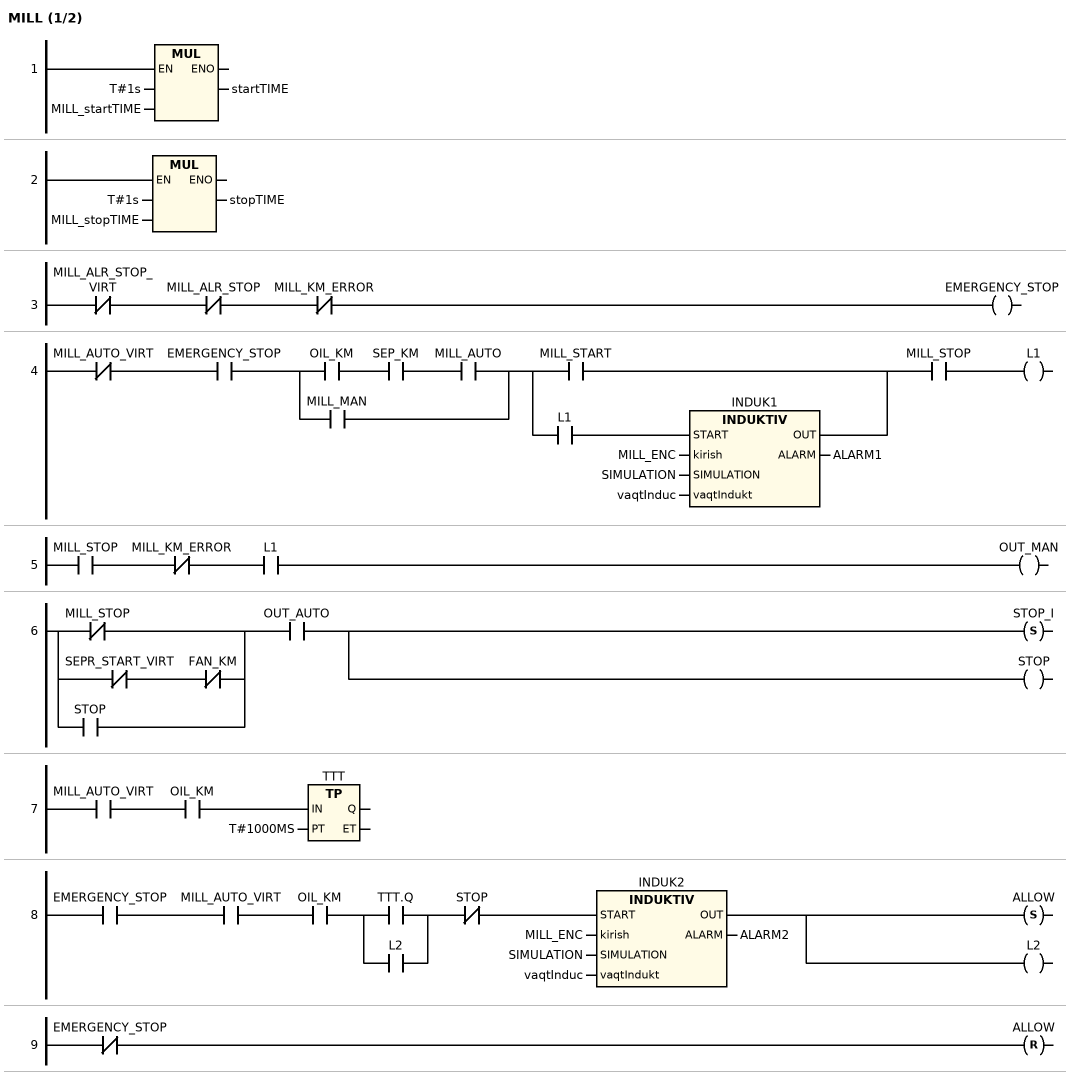
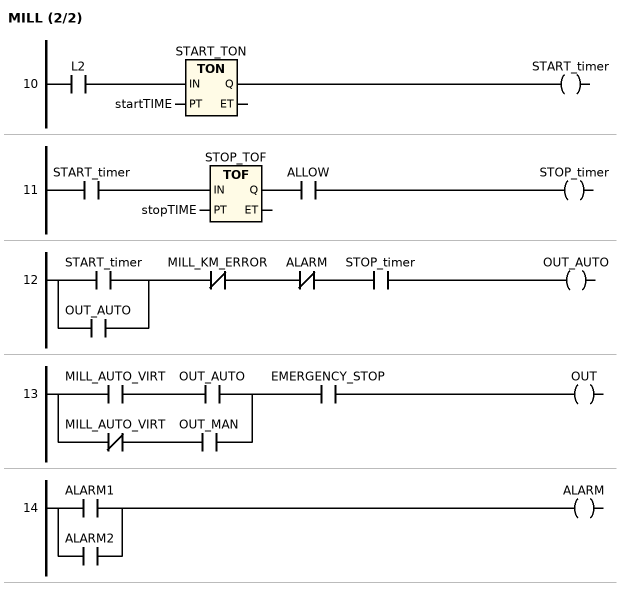
_LD_ (* Ladder Diagram *)
NETWORK 1
	*
		EN --- MUL(T#1s, MILL_startTIME) => startTIME
NETWORK 2
	*
		EN --- MUL(T#1s, MILL_stopTIME) => stopTIME
NETWORK 3
	[/MILL_ALR_STOP_VIRT] - [/MILL_ALR_STOP] - [/MILL_KM_ERROR] --- (EMERGENCY_STOP)
NETWORK 4
	[/MILL_AUTO_VIRT] - [EMERGENCY_STOP] - { [OIL_KM] - [SEP_KM] - [MILL_AUTO] | [MILL_MAN] } - { [MILL_START] | [L1] - INDUK1:INDUKTIV(START: *, kirish: MILL_ENC, SIMULATION: SIMULATION, vaqtIndukt: vaqtInduc, ALARM => ALARM1) } - [MILL_STOP] --- (L1)
NETWORK 5
	[MILL_STOP] - [/MILL_KM_ERROR] - [L1] --- (OUT_MAN)
NETWORK 6
	{ [/MILL_STOP] | [/SEPR_START_VIRT] - [/FAN_KM] | [STOP] } - [OUT_AUTO] --- (S STOP_I) (STOP)
NETWORK 7
	[MILL_AUTO_VIRT] - [OIL_KM] - TTT:TP(IN: *, PT: T#1000MS)
NETWORK 8
	[EMERGENCY_STOP] - [MILL_AUTO_VIRT] - [OIL_KM] - { [TTT.Q] | [L2] } - [/STOP] - INDUK2:INDUKTIV(START: *, kirish: MILL_ENC, SIMULATION: SIMULATION, vaqtIndukt: vaqtInduc, ALARM => ALARM2) --- (S ALLOW) (L2)
NETWORK 9
	[/EMERGENCY_STOP] --- (R ALLOW)
NETWORK 10
	[L2] - START_TON:TON(IN: *, PT: startTIME) --- (START_timer)
NETWORK 11
	[START_timer] - STOP_TOF:TOF(IN: *, PT: stopTIME) - [ALLOW] --- (STOP_timer)
NETWORK 12
	{ [START_timer] | [OUT_AUTO] } - [/MILL_KM_ERROR] - [/ALARM] - [STOP_timer] --- (OUT_AUTO)
NETWORK 13
	{ [MILL_AUTO_VIRT] - [OUT_AUTO] | [/MILL_AUTO_VIRT] - [OUT_MAN] } - [EMERGENCY_STOP] --- (OUT)
NETWORK 14
	{ [ALARM1] | [ALARM2] } --- (ALARM)
_END_LD_
(* the same logic as Structured Text *)
(* Network 1 *)
startTIME := T#1s * MILL_startTIME;
(* Network 2 *)
stopTIME := T#1s * MILL_stopTIME;
(* Network 3 *)
EMERGENCY_STOP := NOT MILL_ALR_STOP_VIRT AND NOT MILL_ALR_STOP AND NOT MILL_KM_ERROR;
(* Network 4 *)
_p1 := NOT MILL_AUTO_VIRT AND EMERGENCY_STOP AND (OIL_KM AND SEP_KM AND MILL_AUTO OR MILL_MAN);
INDUK1(START := _p1 AND L1, kirish := MILL_ENC, SIMULATION := SIMULATION, vaqtIndukt := vaqtInduc);
ALARM1 := INDUK1.ALARM;
L1 := (_p1 AND MILL_START OR INDUK1.OUT) AND MILL_STOP;
(* Network 5 *)
OUT_MAN := MILL_STOP AND NOT MILL_KM_ERROR AND L1;
(* Network 6 *)
_p2 := (NOT MILL_STOP OR NOT SEPR_START_VIRT AND NOT FAN_KM OR STOP) AND OUT_AUTO;
IF _p2 THEN STOP_I := TRUE; END_IF;
STOP := _p2;
(* Network 7 *)
TTT(IN := MILL_AUTO_VIRT AND OIL_KM, PT := T#1000MS);
(* Network 8 *)
INDUK2(START := EMERGENCY_STOP AND MILL_AUTO_VIRT AND OIL_KM AND (TTT.Q OR L2) AND NOT STOP, kirish := MILL_ENC, SIMULATION := SIMULATION, vaqtIndukt := vaqtInduc);
ALARM2 := INDUK2.ALARM;
IF INDUK2.OUT THEN ALLOW := TRUE; END_IF;
L2 := INDUK2.OUT;
(* Network 9 *)
IF NOT EMERGENCY_STOP THEN ALLOW := FALSE; END_IF;
(* Network 10 *)
START_TON(IN := L2, PT := startTIME);
START_timer := START_TON.Q;
(* Network 11 *)
STOP_TOF(IN := START_timer, PT := stopTIME);
STOP_timer := STOP_TOF.Q AND ALLOW;
(* Network 12 *)
OUT_AUTO := (START_timer OR OUT_AUTO) AND NOT MILL_KM_ERROR AND NOT ALARM AND STOP_timer;
(* Network 13 *)
OUT := (MILL_AUTO_VIRT AND OUT_AUTO OR NOT MILL_AUTO_VIRT AND OUT_MAN) AND EMERGENCY_STOP;
(* Network 14 *)
ALARM := ALARM1 OR ALARM2;
END_FUNCTION_BLOCK

(* POU FAN, LD *)
FUNCTION_BLOCK FAN
VAR_INPUT
	EN : BOOL;
	MILL_ALR_STOP: BOOL;
	MILL_ALR_STOP_VIRT : BOOL;
	MILL_AUTO : BOOL;
	MILL_AUTO_VIRT : BOOL;
	MILL_MAN : BOOL;
	FAN_START : BOOL;
	VIBRATOR_T : BOOL;

	FAN_STOP : BOOL;
	MILL_KM : BOOL;

	FAN_KM_ERROR : BOOL;
	SEPR_START_VIRT : BOOL;
	FAN_startTIME : WORD;
	FAN_stopTIME : WORD;
END_VAR

VAR_OUTPUT
	OUT : BOOL;
	ALARM : BOOL;
END_VAR
VAR
	INDUK1: INDUKTIV;
	INDUK2: INDUKTIV;
	OUT_MAN: BOOL;
	OUT_AUTO: BOOL;
	START_TON : TON;
	STOP_TOF : TOF;
	startTIME : TIME;
	stopTIME : TIME;
	L1: BOOL;
	L2: BOOL;
	ES: BOOL;
	EMERGENCY_STOP: BOOL;
	ALARM1 : BOOL;
	ALARM2 : BOOL;

	STOP: BOOL;
	ALLOW: BOOL;
	START_timer: BOOL;
	STOP_timer: BOOL;
	TTT : TP;
END_VAR
VAR (* helpers for the ST form of the networks *)
	_p1 : BOOL;
END_VAR
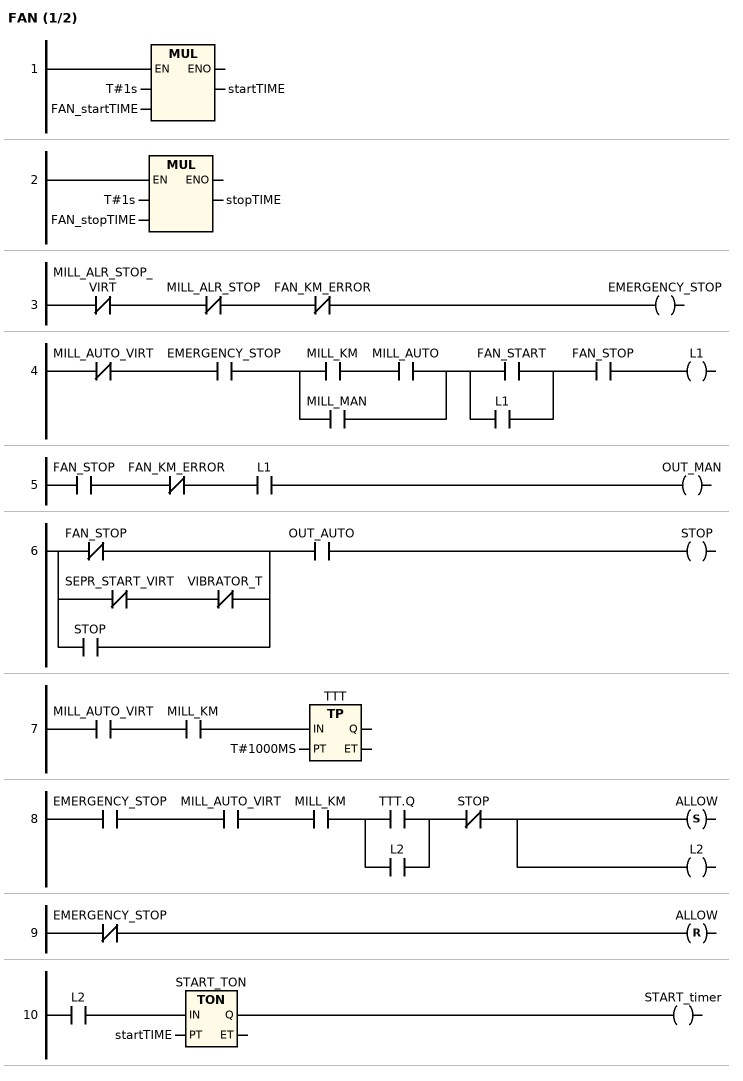
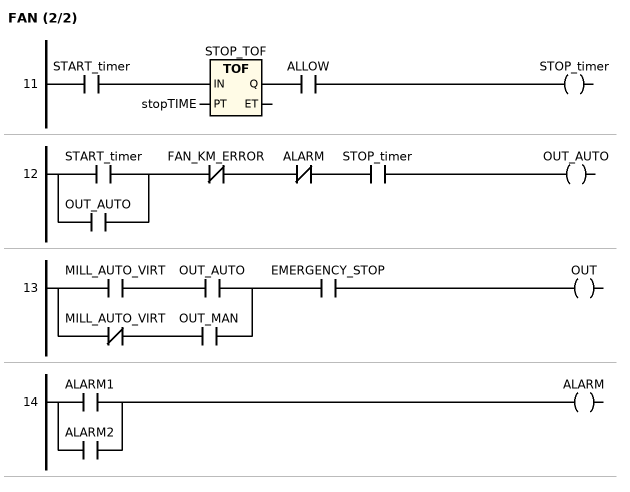
_LD_ (* Ladder Diagram *)
NETWORK 1
	*
		EN --- MUL(T#1s, FAN_startTIME) => startTIME
NETWORK 2
	*
		EN --- MUL(T#1s, FAN_stopTIME) => stopTIME
NETWORK 3
	[/MILL_ALR_STOP_VIRT] - [/MILL_ALR_STOP] - [/FAN_KM_ERROR] --- (EMERGENCY_STOP)
NETWORK 4
	[/MILL_AUTO_VIRT] - [EMERGENCY_STOP] - { [MILL_KM] - [MILL_AUTO] | [MILL_MAN] } - { [FAN_START] | [L1] } - [FAN_STOP] --- (L1)
NETWORK 5
	[FAN_STOP] - [/FAN_KM_ERROR] - [L1] --- (OUT_MAN)
NETWORK 6
	{ [/FAN_STOP] | [/SEPR_START_VIRT] - [/VIBRATOR_T] | [STOP] } - [OUT_AUTO] --- (STOP)
NETWORK 7
	[MILL_AUTO_VIRT] - [MILL_KM] - TTT:TP(IN: *, PT: T#1000MS)
NETWORK 8
	[EMERGENCY_STOP] - [MILL_AUTO_VIRT] - [MILL_KM] - { [TTT.Q] | [L2] } - [/STOP] --- (S ALLOW) (L2)
NETWORK 9
	[/EMERGENCY_STOP] --- (R ALLOW)
NETWORK 10
	[L2] - START_TON:TON(IN: *, PT: startTIME) --- (START_timer)
NETWORK 11
	[START_timer] - STOP_TOF:TOF(IN: *, PT: stopTIME) - [ALLOW] --- (STOP_timer)
NETWORK 12
	{ [START_timer] | [OUT_AUTO] } - [/FAN_KM_ERROR] - [/ALARM] - [STOP_timer] --- (OUT_AUTO)
NETWORK 13
	{ [MILL_AUTO_VIRT] - [OUT_AUTO] | [/MILL_AUTO_VIRT] - [OUT_MAN] } - [EMERGENCY_STOP] --- (OUT)
NETWORK 14
	{ [ALARM1] | [ALARM2] } --- (ALARM)
_END_LD_
(* the same logic as Structured Text *)
(* Network 1 *)
startTIME := T#1s * FAN_startTIME;
(* Network 2 *)
stopTIME := T#1s * FAN_stopTIME;
(* Network 3 *)
EMERGENCY_STOP := NOT MILL_ALR_STOP_VIRT AND NOT MILL_ALR_STOP AND NOT FAN_KM_ERROR;
(* Network 4 *)
L1 := NOT MILL_AUTO_VIRT AND EMERGENCY_STOP AND (MILL_KM AND MILL_AUTO OR MILL_MAN) AND (FAN_START OR L1) AND FAN_STOP;
(* Network 5 *)
OUT_MAN := FAN_STOP AND NOT FAN_KM_ERROR AND L1;
(* Network 6 *)
STOP := (NOT FAN_STOP OR NOT SEPR_START_VIRT AND NOT VIBRATOR_T OR STOP) AND OUT_AUTO;
(* Network 7 *)
TTT(IN := MILL_AUTO_VIRT AND MILL_KM, PT := T#1000MS);
(* Network 8 *)
_p1 := EMERGENCY_STOP AND MILL_AUTO_VIRT AND MILL_KM AND (TTT.Q OR L2) AND NOT STOP;
IF _p1 THEN ALLOW := TRUE; END_IF;
L2 := _p1;
(* Network 9 *)
IF NOT EMERGENCY_STOP THEN ALLOW := FALSE; END_IF;
(* Network 10 *)
START_TON(IN := L2, PT := startTIME);
START_timer := START_TON.Q;
(* Network 11 *)
STOP_TOF(IN := START_timer, PT := stopTIME);
STOP_timer := STOP_TOF.Q AND ALLOW;
(* Network 12 *)
OUT_AUTO := (START_timer OR OUT_AUTO) AND NOT FAN_KM_ERROR AND NOT ALARM AND STOP_timer;
(* Network 13 *)
OUT := (MILL_AUTO_VIRT AND OUT_AUTO OR NOT MILL_AUTO_VIRT AND OUT_MAN) AND EMERGENCY_STOP;
(* Network 14 *)
ALARM := ALARM1 OR ALARM2;
END_FUNCTION_BLOCK

(* POU CONV, LD *)
FUNCTION_BLOCK CONV
VAR_INPUT
	EN : BOOL;
	MILL_ALR_STOP: BOOL;
	MILL_ALR_STOP_VIRT : BOOL;
	MILL_AUTO : BOOL;
	MILL_AUTO_VIRT : BOOL;
	MILL_MAN : BOOL;
	CONV_START : BOOL;
	FAN_KM : BOOL;
	MILL_KM : BOOL;
	CONV_ENC : BOOL;
	CONV_STOP : BOOL;
	VIBRATOR_T : BOOL;
	CONV_KM_ERROR : BOOL;
	SIMULATION : BOOL := TRUE;
	MATER_FULL : BOOL;
	SEPR_START_VIRT : BOOL;
	vaqtInduc : WORD := 15;
END_VAR

VAR_OUTPUT
	OUT : BOOL;
	ALARM : BOOL;
END_VAR
VAR
	INDUK1: INDUKTIV;
	INDUK2: INDUKTIV;
	OUT_MAN: BOOL;
	OUT_AUTO: BOOL;
	START_TON : TON;
	STOP_TOF : TOF;
	startTIME : TIME;
	stopTIME : TIME;
	L1: BOOL;
	L2: BOOL;
	ES: BOOL;
	EMERGENCY_STOP: BOOL;
	ALARM1 : BOOL;
	ALARM2 : BOOL;

	STOP: BOOL;
	ALLOW: BOOL;
	START_timer: BOOL;
	STOP_timer: BOOL;
	TTT : TP;
END_VAR
VAR (* helpers for the ST form of the networks *)
	_p1 : BOOL;
END_VAR
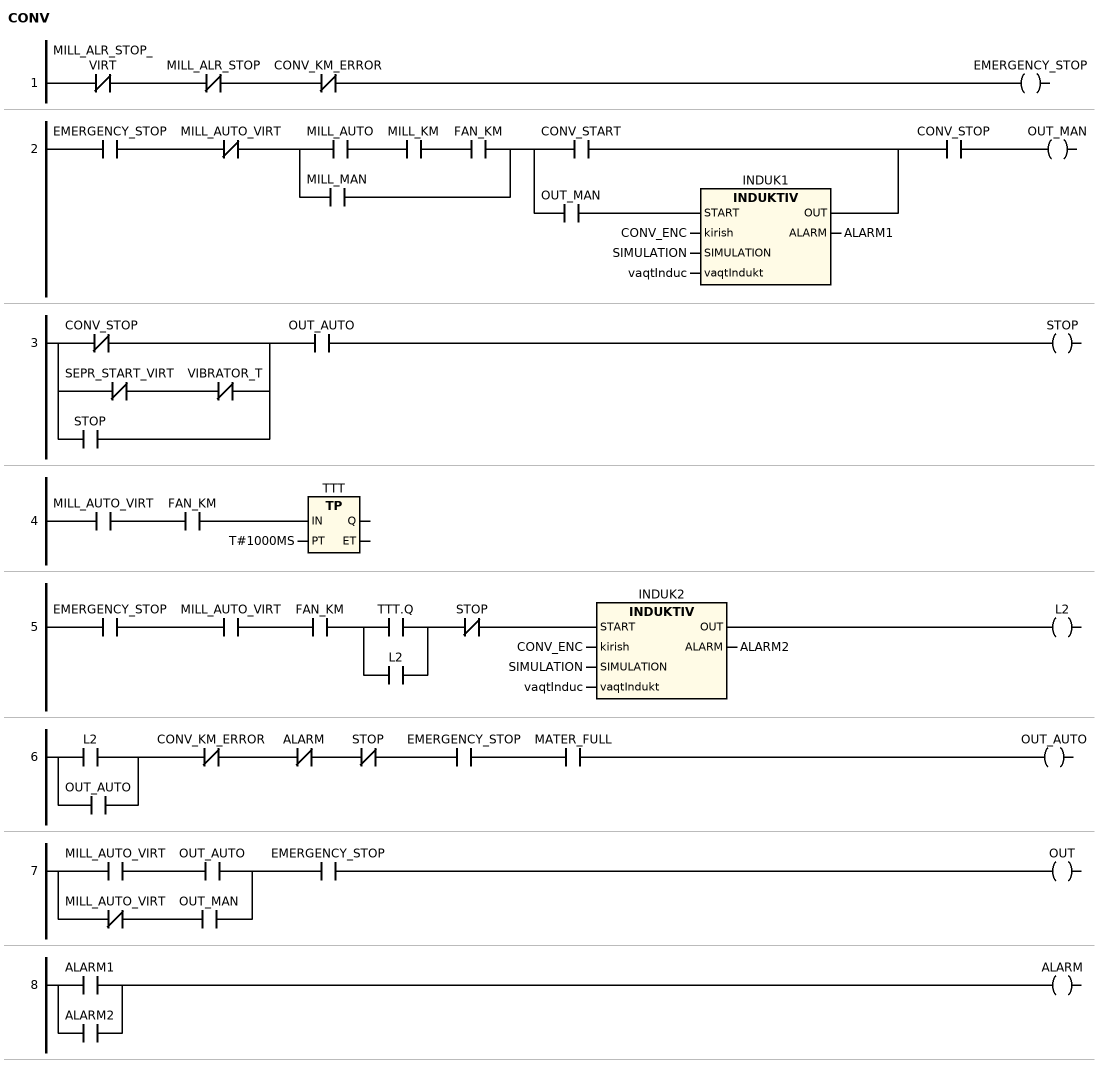
_LD_ (* Ladder Diagram *)
NETWORK 1
	[/MILL_ALR_STOP_VIRT] - [/MILL_ALR_STOP] - [/CONV_KM_ERROR] --- (EMERGENCY_STOP)
NETWORK 2
	[EMERGENCY_STOP] - [/MILL_AUTO_VIRT] - { [MILL_AUTO] - [MILL_KM] - [FAN_KM] | [MILL_MAN] } - { [CONV_START] | [OUT_MAN] - INDUK1:INDUKTIV(START: *, kirish: CONV_ENC, SIMULATION: SIMULATION, vaqtIndukt: vaqtInduc, ALARM => ALARM1) } - [CONV_STOP] --- (OUT_MAN)
NETWORK 3
	{ [/CONV_STOP] | [/SEPR_START_VIRT] - [/VIBRATOR_T] | [STOP] } - [OUT_AUTO] --- (STOP)
NETWORK 4
	[MILL_AUTO_VIRT] - [FAN_KM] - TTT:TP(IN: *, PT: T#1000MS)
NETWORK 5
	[EMERGENCY_STOP] - [MILL_AUTO_VIRT] - [FAN_KM] - { [TTT.Q] | [L2] } - [/STOP] - INDUK2:INDUKTIV(START: *, kirish: CONV_ENC, SIMULATION: SIMULATION, vaqtIndukt: vaqtInduc, ALARM => ALARM2) --- (L2)
NETWORK 6
	{ [L2] | [OUT_AUTO] } - [/CONV_KM_ERROR] - [/ALARM] - [/STOP] - [EMERGENCY_STOP] - [MATER_FULL] --- (OUT_AUTO)
NETWORK 7
	{ [MILL_AUTO_VIRT] - [OUT_AUTO] | [/MILL_AUTO_VIRT] - [OUT_MAN] } - [EMERGENCY_STOP] --- (OUT)
NETWORK 8
	{ [ALARM1] | [ALARM2] } --- (ALARM)
_END_LD_
(* the same logic as Structured Text *)
(* Network 1 *)
EMERGENCY_STOP := NOT MILL_ALR_STOP_VIRT AND NOT MILL_ALR_STOP AND NOT CONV_KM_ERROR;
(* Network 2 *)
_p1 := EMERGENCY_STOP AND NOT MILL_AUTO_VIRT AND (MILL_AUTO AND MILL_KM AND FAN_KM OR MILL_MAN);
INDUK1(START := _p1 AND OUT_MAN, kirish := CONV_ENC, SIMULATION := SIMULATION, vaqtIndukt := vaqtInduc);
ALARM1 := INDUK1.ALARM;
OUT_MAN := (_p1 AND CONV_START OR INDUK1.OUT) AND CONV_STOP;
(* Network 3 *)
STOP := (NOT CONV_STOP OR NOT SEPR_START_VIRT AND NOT VIBRATOR_T OR STOP) AND OUT_AUTO;
(* Network 4 *)
TTT(IN := MILL_AUTO_VIRT AND FAN_KM, PT := T#1000MS);
(* Network 5 *)
INDUK2(START := EMERGENCY_STOP AND MILL_AUTO_VIRT AND FAN_KM AND (TTT.Q OR L2) AND NOT STOP, kirish := CONV_ENC, SIMULATION := SIMULATION, vaqtIndukt := vaqtInduc);
ALARM2 := INDUK2.ALARM;
L2 := INDUK2.OUT;
(* Network 6 *)
OUT_AUTO := (L2 OR OUT_AUTO) AND NOT CONV_KM_ERROR AND NOT ALARM AND NOT STOP AND EMERGENCY_STOP AND MATER_FULL;
(* Network 7 *)
OUT := (MILL_AUTO_VIRT AND OUT_AUTO OR NOT MILL_AUTO_VIRT AND OUT_MAN) AND EMERGENCY_STOP;
(* Network 8 *)
ALARM := ALARM1 OR ALARM2;
END_FUNCTION_BLOCK

(* POU ALARMS, LD *)
PROGRAM ALARMS
VAR
	tofELV: TON;
	tofSHNK3: TON;
	tofSHNK4: TON;
	tofSHNK_SKL_3: TON;
	tofSHNK_SKL_4: TON;
	tofSTAR_31: TON;
	tofSTAR_32: TON;
	tofSTAR_41: TON;
	tofSTAR_42: TON;
	tofSEPR_3: TON;
	tofSEPR_4: TON;
	tofOIL_3: TON;
	tofOIL_4: TON;
	tofMILL_3: TON;
	tofMILL_4: TON;
	tofFAN_3: TON;
	tofFAN_4: TON;
	tofCONV_3: TON;
	tofCONV_4: TON;
	tofVIB_3: TON;
	tofVIB_4: TON;

	vaqt : TIME := T#30S;
END_VAR
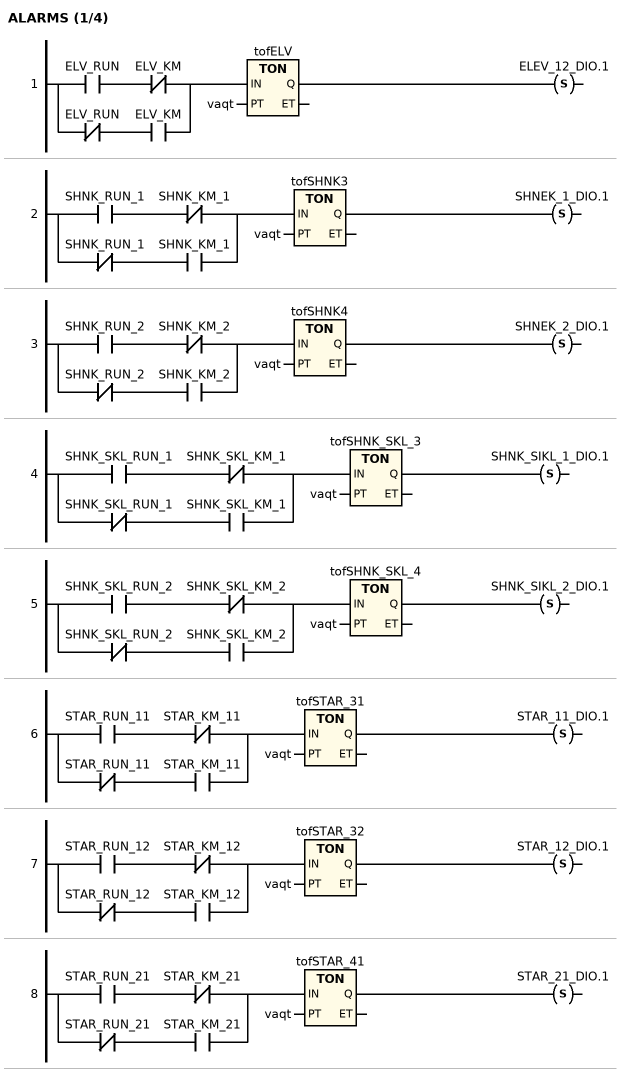
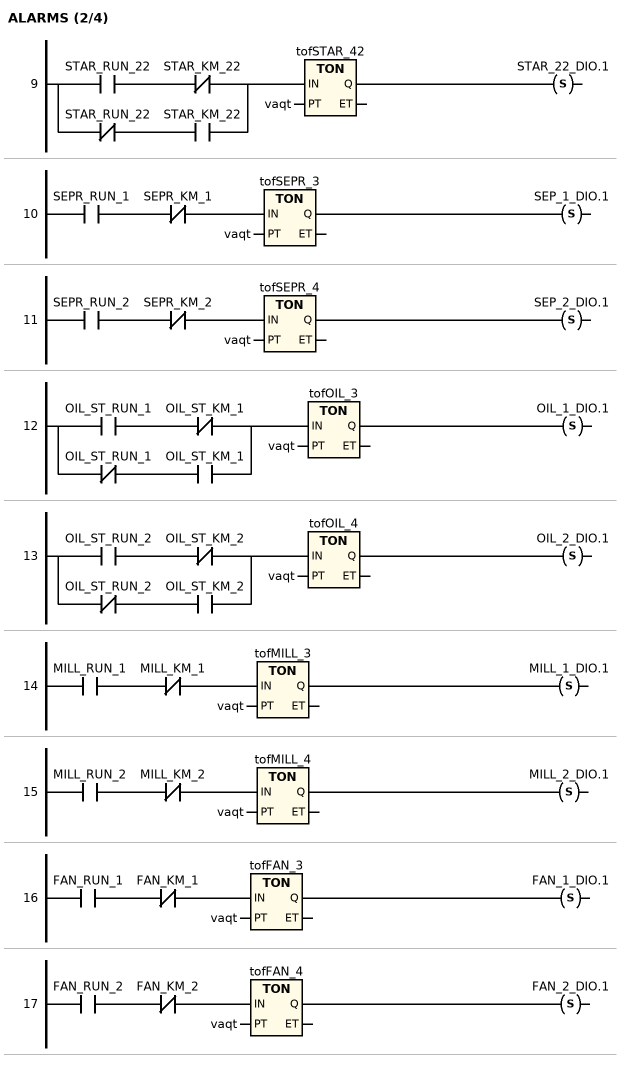
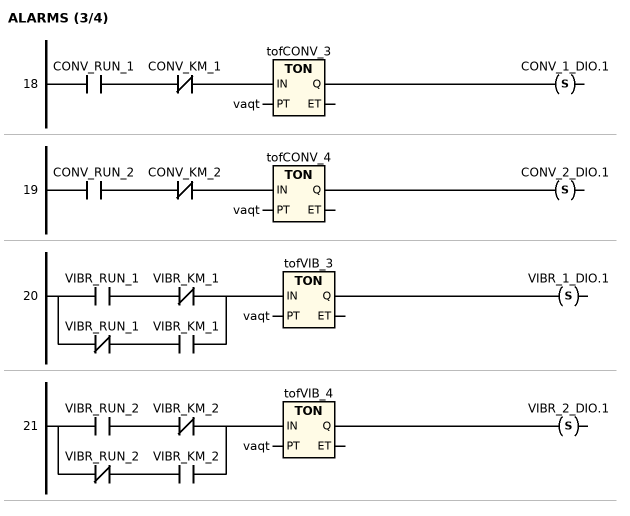
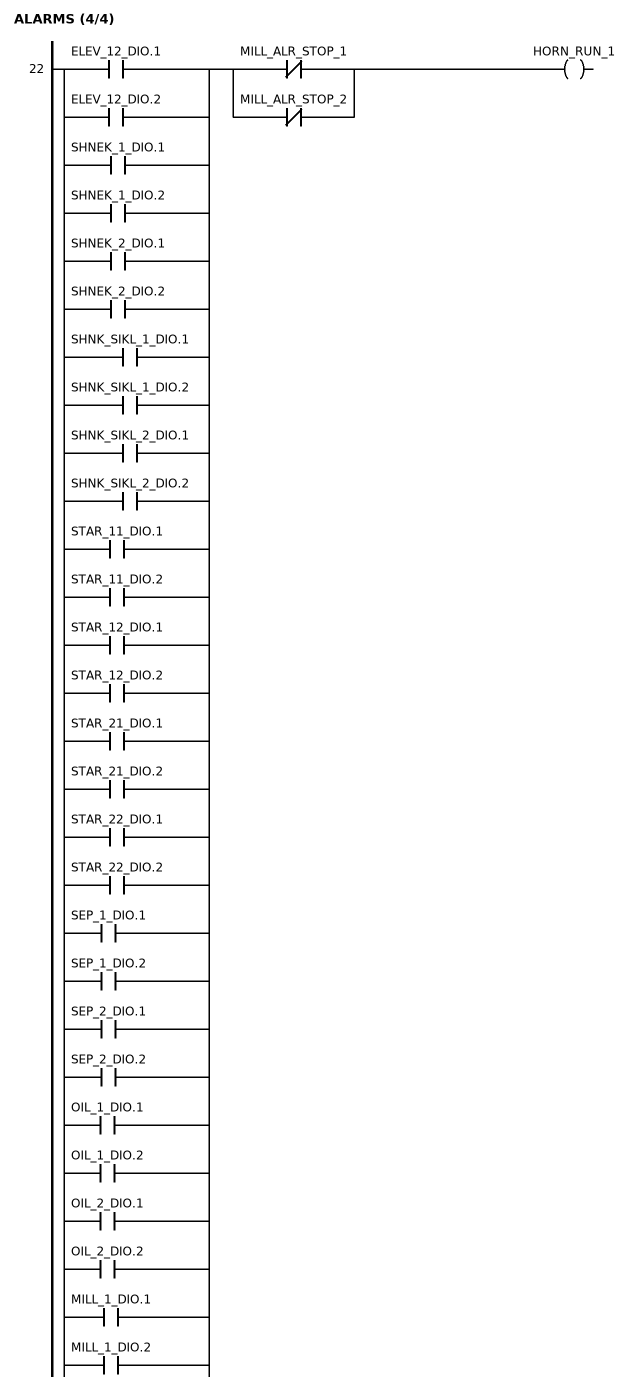
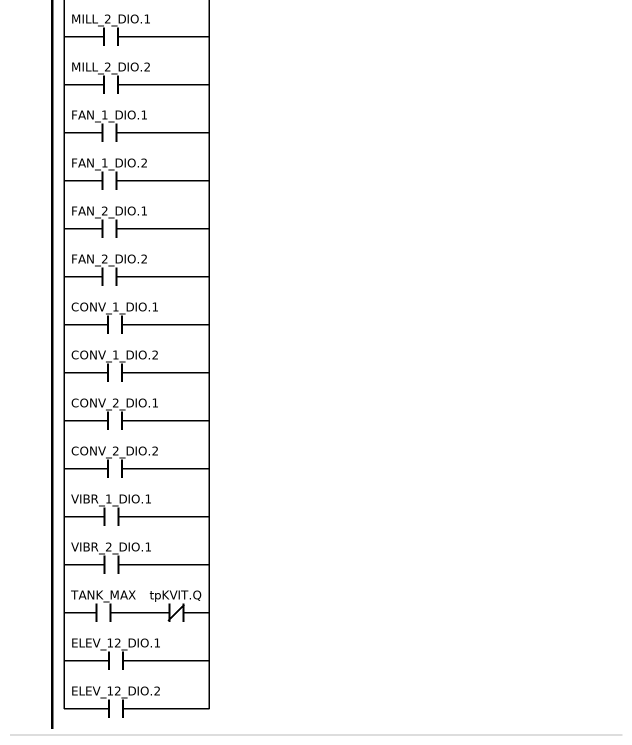
_LD_ (* Ladder Diagram *)
NETWORK 1
	{ [ELV_RUN] - [/ELV_KM] | [/ELV_RUN] - [ELV_KM] } - tofELV:TON(IN: *, PT: vaqt) --- (S ELEV_12_DIO.1)
NETWORK 2
	{ [SHNK_RUN_1] - [/SHNK_KM_1] | [/SHNK_RUN_1] - [SHNK_KM_1] } - tofSHNK3:TON(IN: *, PT: vaqt) --- (S SHNEK_1_DIO.1)
NETWORK 3
	{ [SHNK_RUN_2] - [/SHNK_KM_2] | [/SHNK_RUN_2] - [SHNK_KM_2] } - tofSHNK4:TON(IN: *, PT: vaqt) --- (S SHNEK_2_DIO.1)
NETWORK 4
	{ [SHNK_SKL_RUN_1] - [/SHNK_SKL_KM_1] | [/SHNK_SKL_RUN_1] - [SHNK_SKL_KM_1] } - tofSHNK_SKL_3:TON(IN: *, PT: vaqt) --- (S SHNK_SIKL_1_DIO.1)
NETWORK 5
	{ [SHNK_SKL_RUN_2] - [/SHNK_SKL_KM_2] | [/SHNK_SKL_RUN_2] - [SHNK_SKL_KM_2] } - tofSHNK_SKL_4:TON(IN: *, PT: vaqt) --- (S SHNK_SIKL_2_DIO.1)
NETWORK 6
	{ [STAR_RUN_11] - [/STAR_KM_11] | [/STAR_RUN_11] - [STAR_KM_11] } - tofSTAR_31:TON(IN: *, PT: vaqt) --- (S STAR_11_DIO.1)
NETWORK 7
	{ [STAR_RUN_12] - [/STAR_KM_12] | [/STAR_RUN_12] - [STAR_KM_12] } - tofSTAR_32:TON(IN: *, PT: vaqt) --- (S STAR_12_DIO.1)
NETWORK 8
	{ [STAR_RUN_21] - [/STAR_KM_21] | [/STAR_RUN_21] - [STAR_KM_21] } - tofSTAR_41:TON(IN: *, PT: vaqt) --- (S STAR_21_DIO.1)
NETWORK 9
	{ [STAR_RUN_22] - [/STAR_KM_22] | [/STAR_RUN_22] - [STAR_KM_22] } - tofSTAR_42:TON(IN: *, PT: vaqt) --- (S STAR_22_DIO.1)
NETWORK 10
	[SEPR_RUN_1] - [/SEPR_KM_1] - tofSEPR_3:TON(IN: *, PT: vaqt) --- (S SEP_1_DIO.1)
NETWORK 11
	[SEPR_RUN_2] - [/SEPR_KM_2] - tofSEPR_4:TON(IN: *, PT: vaqt) --- (S SEP_2_DIO.1)
NETWORK 12
	{ [OIL_ST_RUN_1] - [/OIL_ST_KM_1] | [/OIL_ST_RUN_1] - [OIL_ST_KM_1] } - tofOIL_3:TON(IN: *, PT: vaqt) --- (S OIL_1_DIO.1)
NETWORK 13
	{ [OIL_ST_RUN_2] - [/OIL_ST_KM_2] | [/OIL_ST_RUN_2] - [OIL_ST_KM_2] } - tofOIL_4:TON(IN: *, PT: vaqt) --- (S OIL_2_DIO.1)
NETWORK 14
	[MILL_RUN_1] - [/MILL_KM_1] - tofMILL_3:TON(IN: *, PT: vaqt) --- (S MILL_1_DIO.1)
NETWORK 15
	[MILL_RUN_2] - [/MILL_KM_2] - tofMILL_4:TON(IN: *, PT: vaqt) --- (S MILL_2_DIO.1)
NETWORK 16
	[FAN_RUN_1] - [/FAN_KM_1] - tofFAN_3:TON(IN: *, PT: vaqt) --- (S FAN_1_DIO.1)
NETWORK 17
	[FAN_RUN_2] - [/FAN_KM_2] - tofFAN_4:TON(IN: *, PT: vaqt) --- (S FAN_2_DIO.1)
NETWORK 18
	[CONV_RUN_1] - [/CONV_KM_1] - tofCONV_3:TON(IN: *, PT: vaqt) --- (S CONV_1_DIO.1)
NETWORK 19
	[CONV_RUN_2] - [/CONV_KM_2] - tofCONV_4:TON(IN: *, PT: vaqt) --- (S CONV_2_DIO.1)
NETWORK 20
	{ [VIBR_RUN_1] - [/VIBR_KM_1] | [/VIBR_RUN_1] - [VIBR_KM_1] } - tofVIB_3:TON(IN: *, PT: vaqt) --- (S VIBR_1_DIO.1)
NETWORK 21
	{ [VIBR_RUN_2] - [/VIBR_KM_2] | [/VIBR_RUN_2] - [VIBR_KM_2] } - tofVIB_4:TON(IN: *, PT: vaqt) --- (S VIBR_2_DIO.1)
NETWORK 22
	{ [ELEV_12_DIO.1] | [ELEV_12_DIO.2] | [SHNEK_1_DIO.1] | [SHNEK_1_DIO.2] | [SHNEK_2_DIO.1] | [SHNEK_2_DIO.2] | [SHNK_SIKL_1_DIO.1] | [SHNK_SIKL_1_DIO.2] | [SHNK_SIKL_2_DIO.1] | [SHNK_SIKL_2_DIO.2] | [STAR_11_DIO.1] | [STAR_11_DIO.2] | [STAR_12_DIO.1] | [STAR_12_DIO.2] | [STAR_21_DIO.1] | [STAR_21_DIO.2] | [STAR_22_DIO.1] | [STAR_22_DIO.2] | [SEP_1_DIO.1] | [SEP_1_DIO.2] | [SEP_2_DIO.1] | [SEP_2_DIO.2] | [OIL_1_DIO.1] | [OIL_1_DIO.2] | [OIL_2_DIO.1] | [OIL_2_DIO.2] | [MILL_1_DIO.1] | [MILL_1_DIO.2] | [MILL_2_DIO.1] | [MILL_2_DIO.2] | [FAN_1_DIO.1] | [FAN_1_DIO.2] | [FAN_2_DIO.1] | [FAN_2_DIO.2] | [CONV_1_DIO.1] | [CONV_1_DIO.2] | [CONV_2_DIO.1] | [CONV_2_DIO.2] | [VIBR_1_DIO.1] | [VIBR_2_DIO.1] | [TANK_MAX] - [/tpKVIT.Q] | [ELEV_12_DIO.1] | [ELEV_12_DIO.2] } - { [/MILL_ALR_STOP_1] | [/MILL_ALR_STOP_2] } --- (HORN_RUN_1)
_END_LD_
(* the same logic as Structured Text *)
(* Network 1 *)
tofELV(IN := ELV_RUN AND NOT ELV_KM OR NOT ELV_RUN AND ELV_KM, PT := vaqt);
IF tofELV.Q THEN ELEV_12_DIO.1 := TRUE; END_IF;
(* Network 2 *)
tofSHNK3(IN := SHNK_RUN_1 AND NOT SHNK_KM_1 OR NOT SHNK_RUN_1 AND SHNK_KM_1, PT := vaqt);
IF tofSHNK3.Q THEN SHNEK_1_DIO.1 := TRUE; END_IF;
(* Network 3 *)
tofSHNK4(IN := SHNK_RUN_2 AND NOT SHNK_KM_2 OR NOT SHNK_RUN_2 AND SHNK_KM_2, PT := vaqt);
IF tofSHNK4.Q THEN SHNEK_2_DIO.1 := TRUE; END_IF;
(* Network 4 *)
tofSHNK_SKL_3(IN := SHNK_SKL_RUN_1 AND NOT SHNK_SKL_KM_1 OR NOT SHNK_SKL_RUN_1 AND SHNK_SKL_KM_1, PT := vaqt);
IF tofSHNK_SKL_3.Q THEN SHNK_SIKL_1_DIO.1 := TRUE; END_IF;
(* Network 5 *)
tofSHNK_SKL_4(IN := SHNK_SKL_RUN_2 AND NOT SHNK_SKL_KM_2 OR NOT SHNK_SKL_RUN_2 AND SHNK_SKL_KM_2, PT := vaqt);
IF tofSHNK_SKL_4.Q THEN SHNK_SIKL_2_DIO.1 := TRUE; END_IF;
(* Network 6 *)
tofSTAR_31(IN := STAR_RUN_11 AND NOT STAR_KM_11 OR NOT STAR_RUN_11 AND STAR_KM_11, PT := vaqt);
IF tofSTAR_31.Q THEN STAR_11_DIO.1 := TRUE; END_IF;
(* Network 7 *)
tofSTAR_32(IN := STAR_RUN_12 AND NOT STAR_KM_12 OR NOT STAR_RUN_12 AND STAR_KM_12, PT := vaqt);
IF tofSTAR_32.Q THEN STAR_12_DIO.1 := TRUE; END_IF;
(* Network 8 *)
tofSTAR_41(IN := STAR_RUN_21 AND NOT STAR_KM_21 OR NOT STAR_RUN_21 AND STAR_KM_21, PT := vaqt);
IF tofSTAR_41.Q THEN STAR_21_DIO.1 := TRUE; END_IF;
(* Network 9 *)
tofSTAR_42(IN := STAR_RUN_22 AND NOT STAR_KM_22 OR NOT STAR_RUN_22 AND STAR_KM_22, PT := vaqt);
IF tofSTAR_42.Q THEN STAR_22_DIO.1 := TRUE; END_IF;
(* Network 10 *)
tofSEPR_3(IN := SEPR_RUN_1 AND NOT SEPR_KM_1, PT := vaqt);
IF tofSEPR_3.Q THEN SEP_1_DIO.1 := TRUE; END_IF;
(* Network 11 *)
tofSEPR_4(IN := SEPR_RUN_2 AND NOT SEPR_KM_2, PT := vaqt);
IF tofSEPR_4.Q THEN SEP_2_DIO.1 := TRUE; END_IF;
(* Network 12 *)
tofOIL_3(IN := OIL_ST_RUN_1 AND NOT OIL_ST_KM_1 OR NOT OIL_ST_RUN_1 AND OIL_ST_KM_1, PT := vaqt);
IF tofOIL_3.Q THEN OIL_1_DIO.1 := TRUE; END_IF;
(* Network 13 *)
tofOIL_4(IN := OIL_ST_RUN_2 AND NOT OIL_ST_KM_2 OR NOT OIL_ST_RUN_2 AND OIL_ST_KM_2, PT := vaqt);
IF tofOIL_4.Q THEN OIL_2_DIO.1 := TRUE; END_IF;
(* Network 14 *)
tofMILL_3(IN := MILL_RUN_1 AND NOT MILL_KM_1, PT := vaqt);
IF tofMILL_3.Q THEN MILL_1_DIO.1 := TRUE; END_IF;
(* Network 15 *)
tofMILL_4(IN := MILL_RUN_2 AND NOT MILL_KM_2, PT := vaqt);
IF tofMILL_4.Q THEN MILL_2_DIO.1 := TRUE; END_IF;
(* Network 16 *)
tofFAN_3(IN := FAN_RUN_1 AND NOT FAN_KM_1, PT := vaqt);
IF tofFAN_3.Q THEN FAN_1_DIO.1 := TRUE; END_IF;
(* Network 17 *)
tofFAN_4(IN := FAN_RUN_2 AND NOT FAN_KM_2, PT := vaqt);
IF tofFAN_4.Q THEN FAN_2_DIO.1 := TRUE; END_IF;
(* Network 18 *)
tofCONV_3(IN := CONV_RUN_1 AND NOT CONV_KM_1, PT := vaqt);
IF tofCONV_3.Q THEN CONV_1_DIO.1 := TRUE; END_IF;
(* Network 19 *)
tofCONV_4(IN := CONV_RUN_2 AND NOT CONV_KM_2, PT := vaqt);
IF tofCONV_4.Q THEN CONV_2_DIO.1 := TRUE; END_IF;
(* Network 20 *)
tofVIB_3(IN := VIBR_RUN_1 AND NOT VIBR_KM_1 OR NOT VIBR_RUN_1 AND VIBR_KM_1, PT := vaqt);
IF tofVIB_3.Q THEN VIBR_1_DIO.1 := TRUE; END_IF;
(* Network 21 *)
tofVIB_4(IN := VIBR_RUN_2 AND NOT VIBR_KM_2 OR NOT VIBR_RUN_2 AND VIBR_KM_2, PT := vaqt);
IF tofVIB_4.Q THEN VIBR_2_DIO.1 := TRUE; END_IF;
(* Network 22 *)
HORN_RUN_1 := (ELEV_12_DIO.1 OR ELEV_12_DIO.2 OR SHNEK_1_DIO.1 OR SHNEK_1_DIO.2 OR SHNEK_2_DIO.1 OR SHNEK_2_DIO.2 OR SHNK_SIKL_1_DIO.1 OR SHNK_SIKL_1_DIO.2 OR SHNK_SIKL_2_DIO.1 OR SHNK_SIKL_2_DIO.2 OR STAR_11_DIO.1 OR STAR_11_DIO.2 OR STAR_12_DIO.1 OR STAR_12_DIO.2 OR STAR_21_DIO.1 OR STAR_21_DIO.2 OR STAR_22_DIO.1 OR STAR_22_DIO.2 OR SEP_1_DIO.1 OR SEP_1_DIO.2 OR SEP_2_DIO.1 OR SEP_2_DIO.2 OR OIL_1_DIO.1 OR OIL_1_DIO.2 OR OIL_2_DIO.1 OR OIL_2_DIO.2 OR MILL_1_DIO.1 OR MILL_1_DIO.2 OR MILL_2_DIO.1 OR MILL_2_DIO.2 OR FAN_1_DIO.1 OR FAN_1_DIO.2 OR FAN_2_DIO.1 OR FAN_2_DIO.2 OR CONV_1_DIO.1 OR CONV_1_DIO.2 OR CONV_2_DIO.1 OR CONV_2_DIO.2 OR VIBR_1_DIO.1 OR VIBR_2_DIO.1 OR TANK_MAX AND NOT tpKVIT.Q OR ELEV_12_DIO.1 OR ELEV_12_DIO.2) AND (NOT MILL_ALR_STOP_1 OR NOT MILL_ALR_STOP_2);
END_PROGRAM

(* POU RESET_ALRM, LD *)
PROGRAM RESET_ALRM
VAR
END_VAR
VAR (* helpers for the ST form of the networks *)
	_p1 : BOOL;
END_VAR
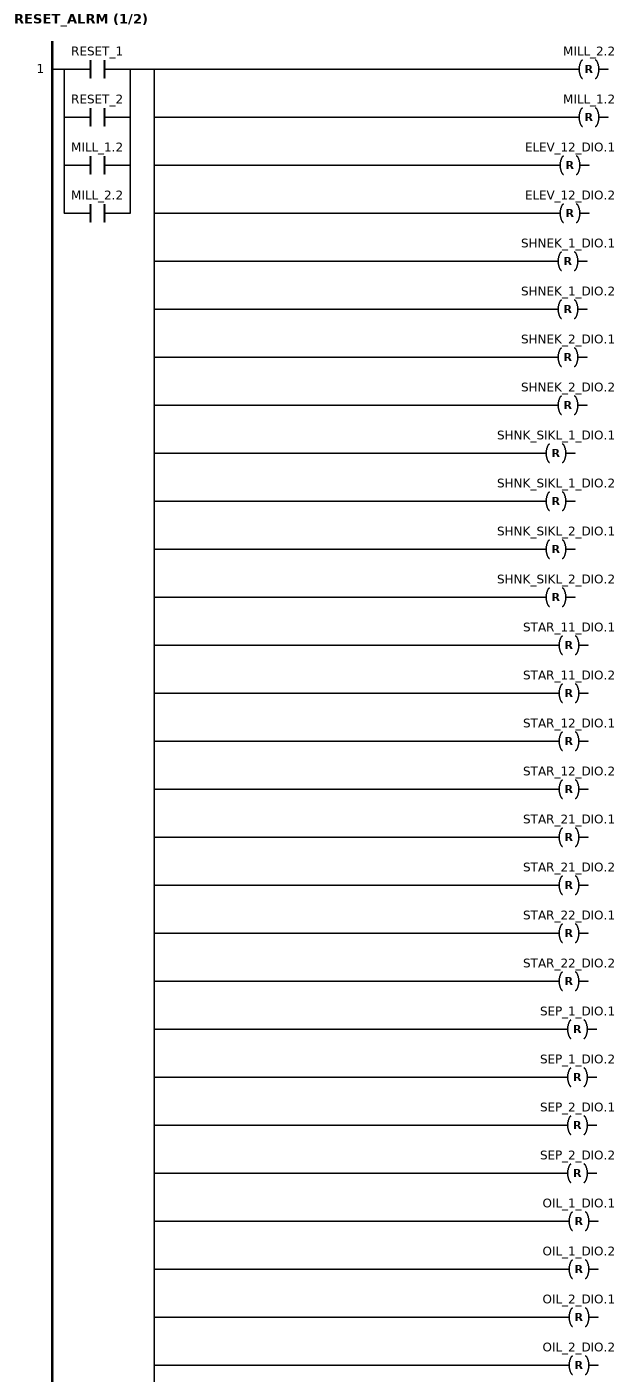
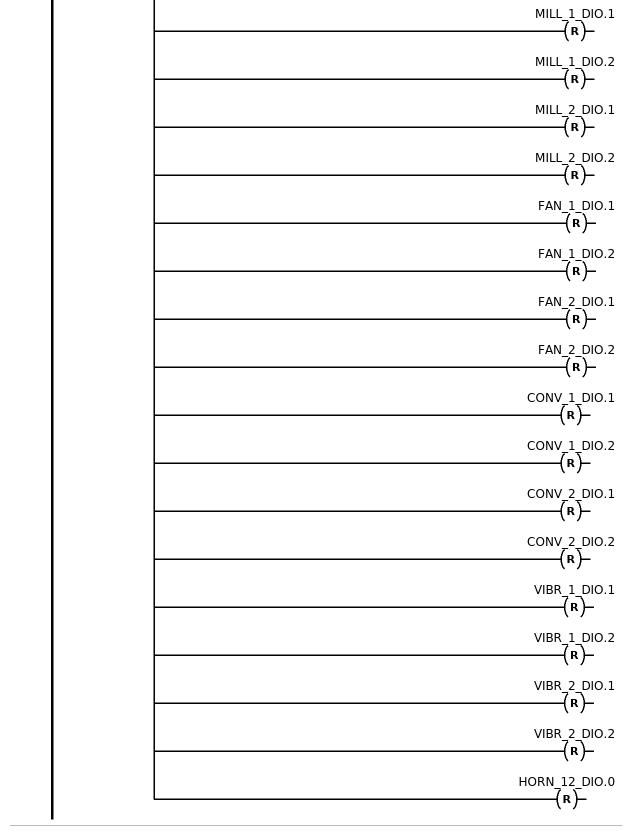
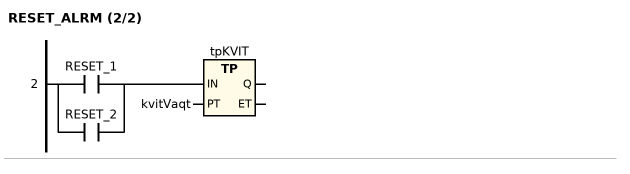
_LD_ (* Ladder Diagram *)
NETWORK 1
	{ [RESET_1] | [RESET_2] | [MILL_1.2] | [MILL_2.2] } --- (R MILL_2.2) (R MILL_1.2) (R ELEV_12_DIO.1) (R ELEV_12_DIO.2) (R SHNEK_1_DIO.1) (R SHNEK_1_DIO.2) (R SHNEK_2_DIO.1) (R SHNEK_2_DIO.2) (R SHNK_SIKL_1_DIO.1) (R SHNK_SIKL_1_DIO.2) (R SHNK_SIKL_2_DIO.1) (R SHNK_SIKL_2_DIO.2) (R STAR_11_DIO.1) (R STAR_11_DIO.2) (R STAR_12_DIO.1) (R STAR_12_DIO.2) (R STAR_21_DIO.1) (R STAR_21_DIO.2) (R STAR_22_DIO.1) (R STAR_22_DIO.2) (R SEP_1_DIO.1) (R SEP_1_DIO.2) (R SEP_2_DIO.1) (R SEP_2_DIO.2) (R OIL_1_DIO.1) (R OIL_1_DIO.2) (R OIL_2_DIO.1) (R OIL_2_DIO.2) (R MILL_1_DIO.1) (R MILL_1_DIO.2) (R MILL_2_DIO.1) (R MILL_2_DIO.2) (R FAN_1_DIO.1) (R FAN_1_DIO.2) (R FAN_2_DIO.1) (R FAN_2_DIO.2) (R CONV_1_DIO.1) (R CONV_1_DIO.2) (R CONV_2_DIO.1) (R CONV_2_DIO.2) (R VIBR_1_DIO.1) (R VIBR_1_DIO.2) (R VIBR_2_DIO.1) (R VIBR_2_DIO.2) (R HORN_12_DIO.0)
NETWORK 2
	{ [RESET_1] | [RESET_2] } - tpKVIT:TP(IN: *, PT: kvitVaqt)
_END_LD_
(* the same logic as Structured Text *)
(* Network 1 *)
_p1 := RESET_1 OR RESET_2 OR MILL_1.2 OR MILL_2.2;
IF _p1 THEN MILL_2.2 := FALSE; MILL_1.2 := FALSE; ELEV_12_DIO.1 := FALSE; ELEV_12_DIO.2 := FALSE; SHNEK_1_DIO.1 := FALSE; SHNEK_1_DIO.2 := FALSE; SHNEK_2_DIO.1 := FALSE; SHNEK_2_DIO.2 := FALSE; SHNK_SIKL_1_DIO.1 := FALSE; SHNK_SIKL_1_DIO.2 := FALSE; SHNK_SIKL_2_DIO.1 := FALSE; SHNK_SIKL_2_DIO.2 := FALSE; STAR_11_DIO.1 := FALSE; STAR_11_DIO.2 := FALSE; STAR_12_DIO.1 := FALSE; STAR_12_DIO.2 := FALSE; STAR_21_DIO.1 := FALSE; STAR_21_DIO.2 := FALSE; STAR_22_DIO.1 := FALSE; STAR_22_DIO.2 := FALSE; SEP_1_DIO.1 := FALSE; SEP_1_DIO.2 := FALSE; SEP_2_DIO.1 := FALSE; SEP_2_DIO.2 := FALSE; OIL_1_DIO.1 := FALSE; OIL_1_DIO.2 := FALSE; OIL_2_DIO.1 := FALSE; OIL_2_DIO.2 := FALSE; MILL_1_DIO.1 := FALSE; MILL_1_DIO.2 := FALSE; MILL_2_DIO.1 := FALSE; MILL_2_DIO.2 := FALSE; FAN_1_DIO.1 := FALSE; FAN_1_DIO.2 := FALSE; FAN_2_DIO.1 := FALSE; FAN_2_DIO.2 := FALSE; CONV_1_DIO.1 := FALSE; CONV_1_DIO.2 := FALSE; CONV_2_DIO.1 := FALSE; CONV_2_DIO.2 := FALSE; VIBR_1_DIO.1 := FALSE; VIBR_1_DIO.2 := FALSE; VIBR_2_DIO.1 := FALSE; VIBR_2_DIO.2 := FALSE; HORN_12_DIO.0 := FALSE; END_IF;
(* Network 2 *)
tpKVIT(IN := RESET_1 OR RESET_2, PT := kvitVaqt);
END_PROGRAM

(* POU TRANSLATE, ST *)
PROGRAM TRANSLATE
VAR
	CON1: A_CONVER;
	CON2: A_CONVER;
	CON3: MY_LIN_TRAFO;
	CON4: A_CONVER;
	CON5: MY_LIN_TRAFO;
	tonTank : TON;
	IN_MIN : REAL := 4;
	IN_MAX: REAL := 20;
	OUT_MIN_SEN : REAL := -10;
	OUT_MAX_SEN: REAL := 1;
	OUT_MIN_CUR : REAL := 0;
	OUT_MAX_CUR: REAL := 50;
END_VAR
freqTask();
MB_ANALOG();

hour_MOVE();


MV8();
MV16();
MV24();
MU32_OUT();
workHour();
TANK_12_DIO.0 := TANK_MIN;
TANK_12_DIO.1 := TANK_MIDL;
TANK_12_DIO.2 := TANK_MAX;
tonTank(IN := TANK_MAX_DI, PT := T#10s);
TANK_MAX := tonTank.Q;
END_PROGRAM
ACTION hour_MOVE:
CONV_1_stopTIME := CONV_1_stopTIME_W;
CONV_1_startTIME := CONV_1_startTIME_W;
FAN_1_stopTIME := FAN_1_stopTIME_W;
FAN_1_startTIME := FAN_1_startTIME_W;
MILL_1_stopTIME := MILL_1_stopTIME_W;
MILL_1_startTIME := MILL_1_startTIME_W;
SEP_1_stopTIME := SEP_1_stopTIME_W;
SEP_1_startTIME := SEP_1_startTIME_W;
CONV_2_stopTIME := CONV_2_stopTIME_W;
CONV_2_startTIME := CONV_2_startTIME_W;
FAN_2_stopTIME := FAN_2_stopTIME_W;
FAN_2_startTIME := FAN_2_startTIME_W;
MILL_2_stopTIME := MILL_2_stopTIME_W;
MILL_2_startTIME := MILL_2_startTIME_W;
SEP_2_stopTIME := SEP_2_stopTIME_W;
SEP_2_startTIME:= SEP_2_startTIME_W;
ELEV_12_stopTIME := ELEV_12_stopTIME_W;
ELEV_12_startTIME := ELEV_12_startTIME_W;
SHNEK_1_stopTIME := SHNEK_1_stopTIME_W;
SHNEK_2_stopTIME := SHNEK_2_stopTIME_W;
SHNEK_1_startTIME := SHNEK_1_startTIME_W;
SHNEK_2_startTIME := SHNEK_2_startTIME_W;
STAR_11_stopTIME := STAR_11_stopTIME_W;
STAR_11_startTIME := STAR_11_startTIME_W;
STAR_12_stopTIME := STAR_12_stopTIME_W;
STAR_12_startTIME := STAR_12_startTIME_W;
STAR_21_stopTIME := STAR_21_stopTIME_W;
STAR_21_startTIME := STAR_21_startTIME_W;
STAR_22_stopTIME := STAR_22_stopTIME_W;
STAR_22_startTIME := STAR_22_startTIME_W;
OIL_1_stopTIME := OIL_1_stopTIME_W;
OIL_1_startTIME := OIL_1_startTIME_W;
OIL_2_stopTIME := OIL_2_stopTIME_W;
OIL_2_startTIME := OIL_2_startTIME_W;
SHNK_SIKL_1_stopTIME := SHNK_SIKL_1_stopTIME_W;
SHNK_SIKL_1_startTIME := SHNK_SIKL_1_startTIME_W;
SHNK_SIKL_2_stopTIME := SHNK_SIKL_2_stopTIME_W;
SHNK_SIKL_2_startTIME := SHNK_SIKL_2_startTIME_W;
END_ACTION
ACTION MB_ANALOG:
ELEV_12_CURRENT := ELV_CURRENT_4;
SHNEK_2_CURRENT := SHNK_CURRENT_4;
FAN_2_SUCTION := MILL_SUCTION_4;
SHNEK_1_CURRENT := SHNK_CURRENT_3;
FAN_1_SUCTION := MILL_SUCTION_3;
END_ACTION
ACTION MU32_OUT:
MU01 := BOOL_TO_WORD(ELV_RUN) * 1000;
MU02 := BOOL_TO_WORD(SHNK_RUN_2) * 1000;
MU03 := BOOL_TO_WORD(SHNK_SKL_RUN_2) * 1000;
MU04 := BOOL_TO_WORD(STAR_RUN_21) * 1000;
MU05 := BOOL_TO_WORD(STAR_RUN_22) * 1000;
MU06 := BOOL_TO_WORD(SEPR_RUN_2) * 1000;
MU07 := BOOL_TO_WORD(OIL_ST_RUN_2) * 1000;
MU08 := BOOL_TO_WORD(MILL_RUN_2) * 1000;
MU09 := BOOL_TO_WORD(FAN_RUN_2) * 1000;
MU10 := BOOL_TO_WORD(CONV_RUN_2) * 1000;
MU11 := BOOL_TO_WORD(VIBR_RUN_2) * 1000;
MU12 := BOOL_TO_WORD(VALV_RUN_2) * 1000;
MU13 := BOOL_TO_WORD(HORN_RUN_2) * 1000;
(*
MU14 := BOOL_TO_WORD(m_out14) * 1000;
MU15 := BOOL_TO_WORD(m_out15) * 1000;
MU16 := BOOL_TO_WORD(m_out16) * 1000;
*)
MU17 := BOOL_TO_WORD(ELV_RUN) * 1000;
MU18 := BOOL_TO_WORD(SHNK_RUN_1) * 1000;
MU19 := BOOL_TO_WORD(SHNK_SKL_RUN_1) * 1000;
MU20 := BOOL_TO_WORD(STAR_RUN_11) * 1000;
MU21 := BOOL_TO_WORD(STAR_RUN_12) * 1000;
MU22 := BOOL_TO_WORD(SEPR_RUN_1) * 1000;
MU23 := BOOL_TO_WORD(OIL_ST_RUN_1) * 1000;
MU24 := BOOL_TO_WORD(MILL_RUN_1) * 1000;
MU25 := BOOL_TO_WORD(FAN_RUN_1) * 1000;
MU26 := BOOL_TO_WORD(CONV_RUN_1) * 1000;
MU27 := BOOL_TO_WORD(VIBR_RUN_1) * 1000;
MU28 := BOOL_TO_WORD(VALV_RUN_1) * 1000;
MU29 := BOOL_TO_WORD(HORN_RUN_1) * 1000;
(*
MU30 := BOOL_TO_WORD(m_out30) * 1000;
MU31 := BOOL_TO_WORD(m_out31) * 1000;
MU32 := BOOL_TO_WORD(m_out32) * 1000;
*)
END_ACTION
ACTION MV16:
ELEV_12_DIO.4			 := ELV_STOP_1	 		:= MV16_0.0;
SHNEK_1_DIO.4 			 := SHNK_STOP_1		 := MV16_0.1;
SHNK_SIKL_1_DIO.4		 :=  SHNK_SKL_STOP_1	 := MV16_0.2;
STAR_11_DIO.4			 := STAR_STOP_11		 := MV16_0.3;
STAR_12_DIO.4			 := STAR_STOP_12		 := MV16_0.4;
SEP_1_DIO.4 				 := SEPR_STOP_1		 := MV16_0.5;
OIL_1_DIO.4				 := OIL_ST_STOP_1		 := MV16_0.6;
MILL_1_DIO.4				 := MILL_STOP_1			 := MV16_0.7;
FAN_1_DIO.4				 := FAN_STOP_1			 := MV16_0.8;
CONV_1_DIO.4			 := CONV_STOP_1		 := MV16_0.9;
VIBR_1_DIO.4                     := VIBR_STOP_1			 := MV16_0.10;
(**********************)
ELEV_12_DIO.3			 := ELV_START_1			 := MV16_1.0;
SHNEK_1_DIO.3 			 := SHNK_START_1		 := MV16_1.1;
SHNK_SIKL_1_DIO.3		 := SHNK_SKL_START_1 := MV16_1.2;
STAR_11_DIO.3			 := STAR_START_11		 := MV16_1.3;
STAR_12_DIO.3			 := STAR_START_12		 := MV16_1.4;
SEP_1_DIO.3 				 := SEPR_START_1		 := MV16_1.5;
OIL_1_DIO.3				 := OIL_ST_START_1		 := MV16_1.6;
MILL_1_DIO.3				 := MILL_START_1		 := MV16_1.7;
FAN_1_DIO.3				 := FAN_START_1 			 := MV16_1.8;
CONV_1_DIO.3			 := CONV_START_1 		 := MV16_1.9;
VIBR_1_DIO.3                     := VIBR_START_1		 := MV16_1.10;
END_ACTION
ACTION MV24:
ELV_KM := MV24_0.0;
SHNK_KM_2 := MV24_0.1;
SHNK_SKL_KM_2 := MV24_0.2;
STAR_KM_21 := MV24_0.3;
STAR_KM_22 := MV24_0.4;
SEPR_KM_2 := MV24_0.5;
OIL_ST_KM_2 := MV24_0.6;
MILL_KM_2 := MV24_0.7;
MILL_2_DIO.8 := MATER_FULL_2 := MV24_0.8;
FAN_KM_2 := MV24_0.9;
CONV_KM_2 := MV24_0.10;
VIBR_KM_2 := MV24_0.11;
(*********
ELV_KM_3 := MV24_1.0;*)
SHNK_KM_1 := MV24_1.1;
SHNK_SKL_KM_1 := MV24_1.2;
STAR_KM_11 := MV24_1.3;
STAR_KM_12 := MV24_1.4;
SEPR_KM_1 := MV24_1.5;
OIL_ST_KM_1 := MV24_1.6;
MILL_KM_1 := MV24_1.7;
MILL_1_DIO.8 := MATER_FULL_1 := MV24_1.8;
FAN_KM_1 := MV24_1.9;
CONV_KM_1 := MV24_1.10;
VIBR_KM_1 := MV24_1.11;
END_ACTION
ACTION MV8:
ELV_STOP_2 := MV8_0.0;
SHNK_STOP_2 := MV8_0.1;
SHNK_SKL_STOP_2 := MV8_0.2;


STAR_21_DIO.4 			:= STAR_STOP_21 			:= MV8_0.3;
STAR_22_DIO.4 			:= STAR_STOP_22			 := MV8_0.4;
SEP_2_DIO.4 				 :=SEPR_STOP_2				 := MV8_0.5;
OIL_2_DIO.4				 := OIL_ST_STOP_2			 := MV8_0.6;
MILL_2_DIO.4				 := MILL_STOP_2				 := MV8_0.7;
FAN_2_DIO.4				 := FAN_STOP_2				 := MV8_0.8;
CONV_2_DIO.4			 :=CONV_STOP_2			 := MV8_0.9;
VIBR_2_DIO.4                     := VIBR_STOP_2				 := MV8_0.10;
(**********************)
ELEV_12_DIO.3			 := ELV_START_2				:= MV8_1.0;
SHNEK_2_DIO.3 			 := SHNK_START_2		 	:= MV8_1.1;
SHNK_SIKL_2_DIO.3		 :=  SHNK_SKL_START_2 	:= MV8_1.2;
STAR_21_DIO.3			 := STAR_START_21			 := MV8_1.3;
STAR_22_DIO.3			 := STAR_START_22 			 := MV8_1.4;
SEP_2_DIO.3 				 := SEPR_START_2			 := MV8_1.5;
OIL_2_DIO.3				 := OIL_ST_START_2			 := MV8_1.6;
MILL_2_DIO.3				 := MILL_START_2			 := MV8_1.7;
FAN_2_DIO.3				 := FAN_START_2				 := MV8_1.8;
CONV_2_DIO.3			 := CONV_START_2			 := MV8_1.9;
VIBR_2_DIO.3                     := VIBR_START_2			 := MV8_1.10;
END_ACTION
ACTION TR_REG_1:
(*
REG_1.0 := MB_ELV_ALR;
REG_1.1 := MB_ELV_ALR_ENC;
REG_1.2 := MB_SHNK_ALR_4;
REG_1.3 :=MB_SHNK_ENC_ALR_4 ;
REG_1.4 := MB_SHNK_SKL_ALR_4;
REG_1.5 := MB_SHNK_SKL_ENC_ALR_4;
REG_1.6 :=MB_STAR_ALR_41 ;
REG_1.7 := MB_STAR_ALR_42;

REG_1.8 := MB_SEPR_ALR_4;
REG_1.9 := MB_OIL_ST_ALR_4;
REG_1.10 :=MB_MILL_ALR_4 ;
REG_1.11 := MB_FAN_ALR_4;
REG_1.12 := MB_CONV_ALR_4;
REG_1.13 := MB_VIBR_ALR_4 ;
REG_1.14 := MB_MILL_ENC_ALR_4;
REG_1.15 := MB_SEPR_ENC_ALR_4;
*);
END_ACTION
ACTION TR_REG_2:
(*
REG_2.0 := MB_SHNK_ALR_3;
REG_2.1 := MB_SHNK_ENC_ALR_3;
REG_2.2 := MB_SHNK_SKL_ALR_3;
REG_2.3 := MB_STAR_ALR_31;
REG_2.4 := MB_STAR_ALR_32;
REG_2.5 := MB_SEPR_ALR_3;
REG_2.6 := MB_SEPR_ENC_ALR_3;
REG_2.7 := MB_OIL_ST_ALR_3;

REG_2.8 := MB_MILL_ALR_3;
REG_2.10 := MB_FAN_ALR_3;
REG_2.11 := MB_CONV_ALR_3;
REG_2.12 := MB_VIBR_ALR_3;
REG_2.13 := MB_MILL_ENC_ALR_3;
REG_2.14 := MB_TANK_MIN;
REG_2.15 := MB_TANK_MAX;

*)
;
END_ACTION
ACTION TR_REG_3:
(*
REG_3.0 := MB_ELV_RUN;
REG_3.1 := MB_SHNK_RUN_4;
REG_3.2 := MB_SHNK_SKL_RUN_4;
REG_3.3 := MB_STAR_RUN_41;
REG_3.4 := MB_STAR_RUN_42;
REG_3.5 := MB_SEPR_RUN_4;
REG_3.6 := MB_OIL_ST_RUN_4;
REG_3.7 := MB_MILL_RUN_4;

REG_3.8 := MB_FAN_RUN_4;
REG_3.9 := MB_CONV_RUN_4;
REG_3.10 := MB_VIBR_RUN_4;
REG_3.11 := MB_VALV_RUN_4;
REG_3.12 := MB_HORN_RUN;
REG_3.13 := MB_MATER_FULL_4;

*)
;
END_ACTION
ACTION TR_REG_4:
(*
REG_4.0 := MB_SHNK_RUN_3;
REG_4.1 := MB_SHNK_SKL_RUN_3;
REG_4.2 := MB_STAR_RUN_31;
REG_4.3 := MB_STAR_RUN_32;
REG_4.4 := MB_SEPR_RUN_3;
REG_4.5 := MB_OIL_ST_RUN_3;
REG_4.6 := MB_MILL_RUN_3;
REG_4.7 := MB_FAN_RUN_3;

REG_4.8 := MB_CONV_RUN_3;
REG_4.9 := MB_VIBR_RUN_3;
REG_4.10 := MB_VALV_RUN_3;
REG_4.11 := MB_MATER_FULL_3;

*)
;
END_ACTION

(* POU A_CONVER, CFC *)
FUNCTION_BLOCK A_CONVER
VAR_INPUT
	IN : REAL;
	IN_MIN : REAL := 4;
	IN_MAX : REAL := 20;
	OUT_MIN : REAL := 4;
	OUT_MAX : REAL := 20;
END_VAR
VAR_OUTPUT
	OUT : WORD;

END_VAR
VAR
	LIN1: LIN_TRAFO;
END_VAR
VAR (* helpers for the ST form of the networks *)
	_t11 : WORD;
END_VAR
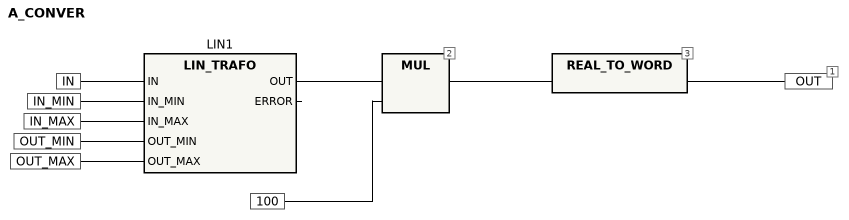
_CFC_ (* Continuous Function Chart, elements in execution order *)
#0 LIN1:LIN_TRAFO(IN: IN, IN_MIN: IN_MIN, IN_MAX: IN_MAX, OUT_MIN: OUT_MIN, OUT_MAX: OUT_MAX)
#1 OUT <= #3
#2 MUL(#0.OUT, 100)
#3 REAL_TO_WORD(#2)
_END_CFC_
(* the same logic as Structured Text *)
LIN1(IN := IN, IN_MIN := IN_MIN, IN_MAX := IN_MAX, OUT_MIN := OUT_MIN, OUT_MAX := OUT_MAX);
OUT := _t11;
_t11 := REAL_TO_WORD(LIN1.OUT * 100);
END_FUNCTION_BLOCK

(* POU MY_LIN_TRAFO, CFC *)
FUNCTION_BLOCK MY_LIN_TRAFO
VAR_INPUT
	IN : REAL;
	IN_MIN : REAL;
	IN_MAX : REAL;
	OUT_MIN : REAL;
	OUT_MAX : REAL;
END_VAR
VAR_OUTPUT
	OUT : REAL;
END_VAR
VAR
	TRA: LIN_TRAFO;
END_VAR
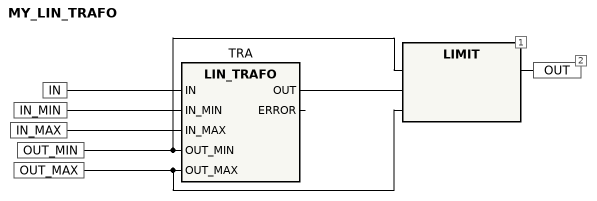
_CFC_ (* Continuous Function Chart, elements in execution order *)
#0 TRA:LIN_TRAFO(IN: IN, IN_MIN: IN_MIN, IN_MAX: IN_MAX, OUT_MIN: OUT_MIN, OUT_MAX: OUT_MAX)
#1 LIMIT(OUT_MIN, #0.OUT, OUT_MAX)
#2 OUT <= #1
_END_CFC_
(* the same logic as Structured Text *)
TRA(IN := IN, IN_MIN := IN_MIN, IN_MAX := IN_MAX, OUT_MIN := OUT_MIN, OUT_MAX := OUT_MAX);
OUT := LIMIT(OUT_MIN, TRA.OUT, OUT_MAX);
END_FUNCTION_BLOCK

(* POU freqTask, ST *)
PROGRAM freqTask
VAR
END_VAR
CONV_1_CURRENT := CONV_CURRENT_1;
CONV_1_FREQ := CONV_FREQ_1;
CONV_SET_FREQ_1 := CONV_1_SETPOINT;

FAN_1_CURRENT :=FAN_CURRENT_1;
FAN_1_FREQ := FAN_FREQ_1;
FAN_SET_FREQ_1 := FAN_1_SETPOINT;

MILL_1_CURRENT :=MILL_CURRENT_1;
MILL_1_FREQ := MILL_FREQ_1;
MILL_SET_FREQ_1 := MILL_1_SETPOINT;

SEP_1_CURRENT :=SEP_CURRENT_1;
SEP_1_FREQ := SEP_FREQ_1;
SEP_SET_FREQ_1 := SEP_1_SETPOINT;

CONV_2_CURRENT := CONV_CURRENT_2;
CONV_2_FREQ := CONV_FREQ_2;
CONV_SET_FREQ_2 := CONV_2_SETPOINT;

FAN_2_CURRENT :=FAN_CURRENT_2;
FAN_2_FREQ := FAN_FREQ_2;
FAN_SET_FREQ_2 := FAN_2_SETPOINT;

MILL_2_CURRENT :=MILL_CURRENT_2;
MILL_2_FREQ := MILL_FREQ_2;
MILL_SET_FREQ_2 := MILL_2_SETPOINT;

SEP_2_CURRENT :=SEP_CURRENT_2;
SEP_2_FREQ := SEP_FREQ_2;
SEP_SET_FREQ_2 := SEP_2_SETPOINT;



IF MILL_1.4 THEN
	CONV_PANEL_1 :=8;
	FAN_PANEL_1 :=9;
	MILL_PANEL_1 :=8;
	SEP_PANEL_1 :=8;
ELSE
	CONV_PANEL_1 :=0;
	FAN_PANEL_1 :=2;
	MILL_PANEL_1 :=0;
	SEP_PANEL_1 :=0;
END_IF;

IF MILL_2.4 THEN
	CONV_PANEL_2 :=8;
	FAN_PANEL_2 :=9;
	MILL_PANEL_2 :=8;
	SEP_PANEL_2 :=8;
ELSE
	CONV_PANEL_2 :=0;
	FAN_PANEL_2 :=2;
	MILL_PANEL_2 :=0;
	SEP_PANEL_2 :=0;
END_IF;
END_PROGRAM

(* POU workHour, LD *)
PROGRAM workHour
VAR
	evlev1_hour : calcHOUR;
	CONV_1_hour : calcHOUR;
	FAN_1_hour : calcHOUR;
	MILL_1_hour : calcHOUR;
	SEP_1_hour : calcHOUR;
	CONV_2_hour : calcHOUR;
	FAN_2_hour : calcHOUR;

	MILL_2_hour: calcHOUR;
	SEP_2_hour: calcHOUR;
	SHNEK_1_hour: calcHOUR;
	SHNEK_2_hour: calcHOUR;
	STAR_11_hour: calcHOUR;
	STAR_12_hour: calcHOUR;
	STAR_21_hour: calcHOUR;
	STAR_22_hour: calcHOUR;
	OIL_1_hour: calcHOUR;
	OIL_2_hour: calcHOUR;
	SHNK_SIKL_1_hour: calcHOUR;
	SHNK_SIKL_2_hour: calcHOUR;

END_VAR
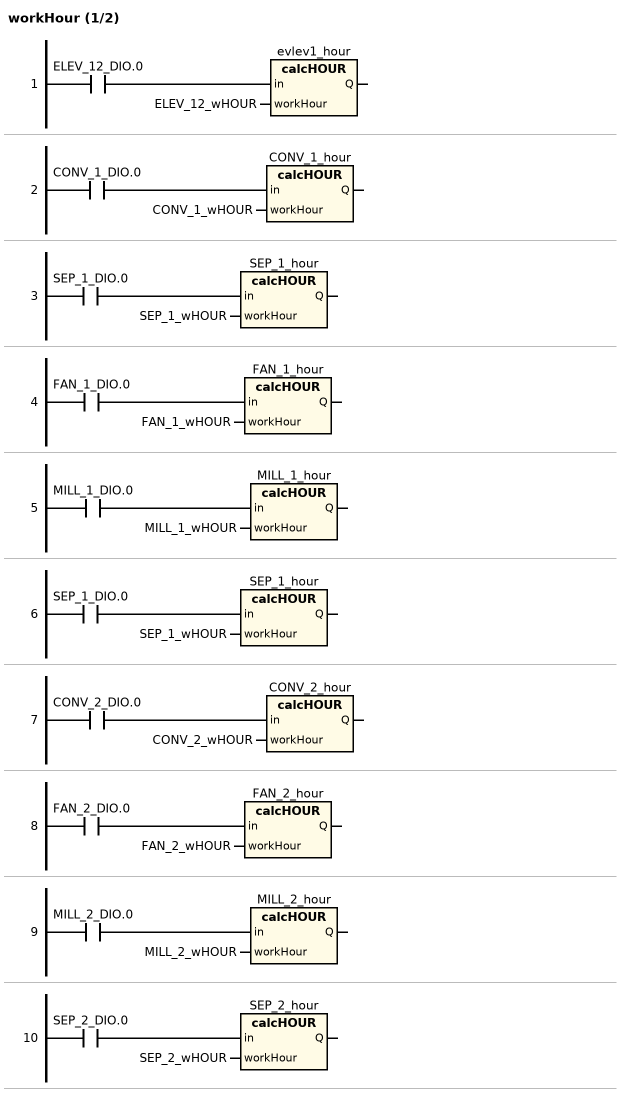
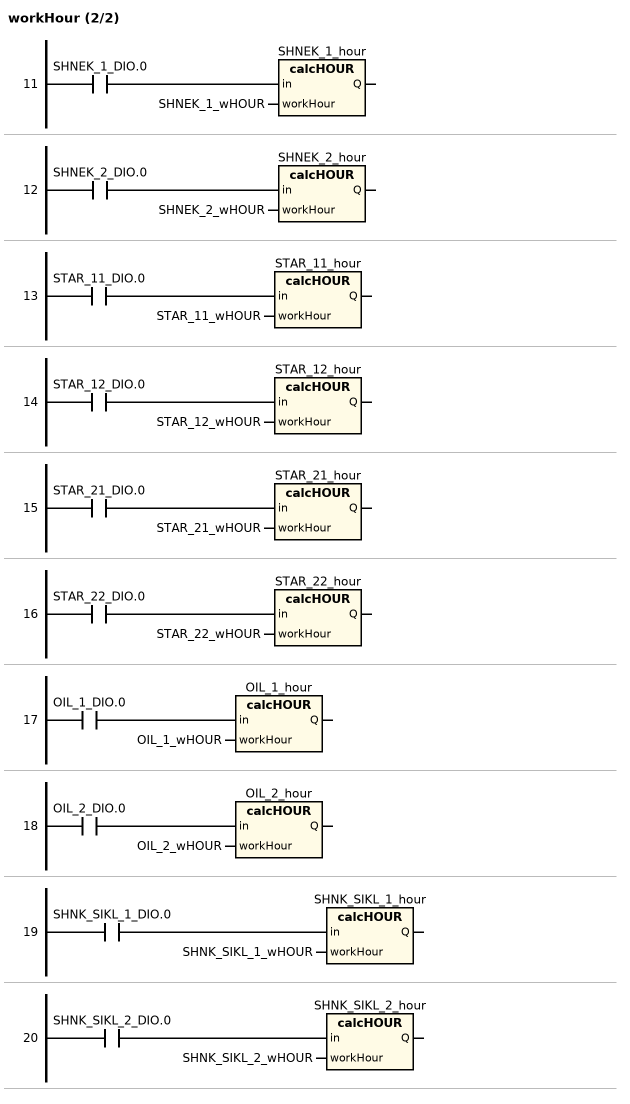
_LD_ (* Ladder Diagram *)
NETWORK 1
	[ELEV_12_DIO.0] - evlev1_hour:calcHOUR(in: *, workHour: ELEV_12_wHOUR)
NETWORK 2
	[CONV_1_DIO.0] - CONV_1_hour:calcHOUR(in: *, workHour: CONV_1_wHOUR)
NETWORK 3
	[SEP_1_DIO.0] - SEP_1_hour:calcHOUR(in: *, workHour: SEP_1_wHOUR)
NETWORK 4
	[FAN_1_DIO.0] - FAN_1_hour:calcHOUR(in: *, workHour: FAN_1_wHOUR)
NETWORK 5
	[MILL_1_DIO.0] - MILL_1_hour:calcHOUR(in: *, workHour: MILL_1_wHOUR)
NETWORK 6
	[SEP_1_DIO.0] - SEP_1_hour:calcHOUR(in: *, workHour: SEP_1_wHOUR)
NETWORK 7
	[CONV_2_DIO.0] - CONV_2_hour:calcHOUR(in: *, workHour: CONV_2_wHOUR)
NETWORK 8
	[FAN_2_DIO.0] - FAN_2_hour:calcHOUR(in: *, workHour: FAN_2_wHOUR)
NETWORK 9
	[MILL_2_DIO.0] - MILL_2_hour:calcHOUR(in: *, workHour: MILL_2_wHOUR)
NETWORK 10
	[SEP_2_DIO.0] - SEP_2_hour:calcHOUR(in: *, workHour: SEP_2_wHOUR)
NETWORK 11
	[SHNEK_1_DIO.0] - SHNEK_1_hour:calcHOUR(in: *, workHour: SHNEK_1_wHOUR)
NETWORK 12
	[SHNEK_2_DIO.0] - SHNEK_2_hour:calcHOUR(in: *, workHour: SHNEK_2_wHOUR)
NETWORK 13
	[STAR_11_DIO.0] - STAR_11_hour:calcHOUR(in: *, workHour: STAR_11_wHOUR)
NETWORK 14
	[STAR_12_DIO.0] - STAR_12_hour:calcHOUR(in: *, workHour: STAR_12_wHOUR)
NETWORK 15
	[STAR_21_DIO.0] - STAR_21_hour:calcHOUR(in: *, workHour: STAR_21_wHOUR)
NETWORK 16
	[STAR_22_DIO.0] - STAR_22_hour:calcHOUR(in: *, workHour: STAR_22_wHOUR)
NETWORK 17
	[OIL_1_DIO.0] - OIL_1_hour:calcHOUR(in: *, workHour: OIL_1_wHOUR)
NETWORK 18
	[OIL_2_DIO.0] - OIL_2_hour:calcHOUR(in: *, workHour: OIL_2_wHOUR)
NETWORK 19
	[SHNK_SIKL_1_DIO.0] - SHNK_SIKL_1_hour:calcHOUR(in: *, workHour: SHNK_SIKL_1_wHOUR)
NETWORK 20
	[SHNK_SIKL_2_DIO.0] - SHNK_SIKL_2_hour:calcHOUR(in: *, workHour: SHNK_SIKL_2_wHOUR)
_END_LD_
(* the same logic as Structured Text *)
(* Network 1 *)
evlev1_hour(in := ELEV_12_DIO.0, workHour := ELEV_12_wHOUR);
(* Network 2 *)
CONV_1_hour(in := CONV_1_DIO.0, workHour := CONV_1_wHOUR);
(* Network 3 *)
SEP_1_hour(in := SEP_1_DIO.0, workHour := SEP_1_wHOUR);
(* Network 4 *)
FAN_1_hour(in := FAN_1_DIO.0, workHour := FAN_1_wHOUR);
(* Network 5 *)
MILL_1_hour(in := MILL_1_DIO.0, workHour := MILL_1_wHOUR);
(* Network 6 *)
SEP_1_hour(in := SEP_1_DIO.0, workHour := SEP_1_wHOUR);
(* Network 7 *)
CONV_2_hour(in := CONV_2_DIO.0, workHour := CONV_2_wHOUR);
(* Network 8 *)
FAN_2_hour(in := FAN_2_DIO.0, workHour := FAN_2_wHOUR);
(* Network 9 *)
MILL_2_hour(in := MILL_2_DIO.0, workHour := MILL_2_wHOUR);
(* Network 10 *)
SEP_2_hour(in := SEP_2_DIO.0, workHour := SEP_2_wHOUR);
(* Network 11 *)
SHNEK_1_hour(in := SHNEK_1_DIO.0, workHour := SHNEK_1_wHOUR);
(* Network 12 *)
SHNEK_2_hour(in := SHNEK_2_DIO.0, workHour := SHNEK_2_wHOUR);
(* Network 13 *)
STAR_11_hour(in := STAR_11_DIO.0, workHour := STAR_11_wHOUR);
(* Network 14 *)
STAR_12_hour(in := STAR_12_DIO.0, workHour := STAR_12_wHOUR);
(* Network 15 *)
STAR_21_hour(in := STAR_21_DIO.0, workHour := STAR_21_wHOUR);
(* Network 16 *)
STAR_22_hour(in := STAR_22_DIO.0, workHour := STAR_22_wHOUR);
(* Network 17 *)
OIL_1_hour(in := OIL_1_DIO.0, workHour := OIL_1_wHOUR);
(* Network 18 *)
OIL_2_hour(in := OIL_2_DIO.0, workHour := OIL_2_wHOUR);
(* Network 19 *)
SHNK_SIKL_1_hour(in := SHNK_SIKL_1_DIO.0, workHour := SHNK_SIKL_1_wHOUR);
(* Network 20 *)
SHNK_SIKL_2_hour(in := SHNK_SIKL_2_DIO.0, workHour := SHNK_SIKL_2_wHOUR);
END_PROGRAM

(* POU calcHOUR, CFC *)
FUNCTION_BLOCK calcHOUR
VAR_INPUT
	in : BOOL;
END_VAR
VAR_IN_OUT
	workHour : WORD;
END_VAR
VAR
	tp1: TP;
	go : BOOL;
	rtrig: R_TRIG;
	ctu1: CTU;
	vaqt : WORD := 3600;
END_VAR
VAR (* helpers for the ST form of the networks *)
	_t14 : WORD;
	_en14 : BOOL;
END_VAR
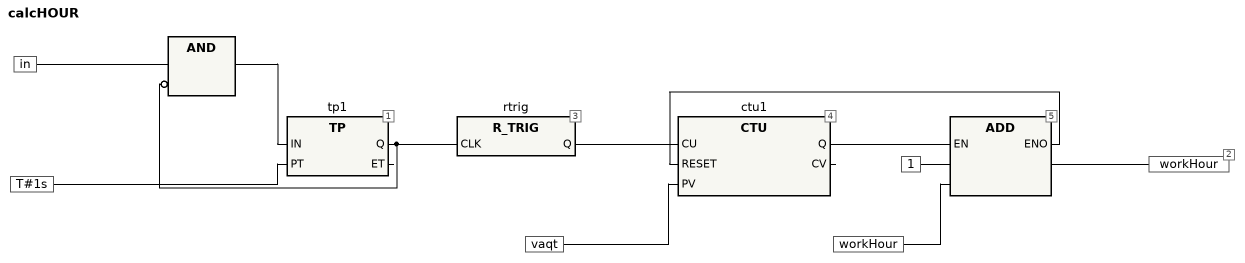
_CFC_ (* Continuous Function Chart, elements in execution order *)
#0 AND(in, NOT #1.Q)
#1 tp1:TP(IN: #0, PT: T#1s)
#2 workHour <= #5
#3 rtrig:R_TRIG(CLK: #1.Q)
#4 ctu1:CTU(CU: #3.Q, RESET: #5.ENO, PV: vaqt)
#5 ADD(EN: #4.Q, 1, workHour)
_END_CFC_
(* the same logic as Structured Text *)
tp1(IN := in AND NOT tp1.Q, PT := T#1s);
workHour := _t14;
rtrig(CLK := tp1.Q);
ctu1(CU := rtrig.Q, RESET := _en14, PV := vaqt);
_en14 := ctu1.Q;
IF _en14 THEN _t14 := 1 + workHour; END_IF;
END_FUNCTION_BLOCK

(* Visualisation TEST
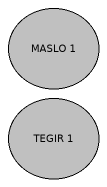
ellipse at (420,440)-(511,521): text "TEGIR 1"; alarm colour if .MILL_RUN_1
ellipse at (420,350)-(511,431): text "MASLO 1"; alarm colour if .MILL_RUN_1
*)
